TYPE PositioningControl :
STRUCT
	Execute : BOOL;
	EmergencyStop : BOOL;
END_STRUCT
END_TYPE

(* stored: Version 1.1.0.1, ProductVersion 3.1.4024.11
   DUT PositioningControl: Id {29284844-ea0e-4aa1-ab50-ccd902667bc2} *)
